TYPE ComplexStruct :
STRUCT
	intVal	:INT:=100;
	DintArr: ARRAY[1..5] OF DINT := [1, 2, 3, 4,100];
	BoolVal	:BOOL:= TRUE;
	ByteVal	:BYTE:=12;
	LrealVal	:LREAL:= 123.67;
	strVal 	:STRING(10):= 'hello';
	//strArray: ARRAY[1..3] OF STRING(10) := ['abc', 'qwe', 'hjk'];  ??
	SimpleStruct1		:SimpleStruct;	
END_STRUCT
END_TYPE

(* stored: Version 1.1.0.1, ProductVersion 3.1.4022.16
   DUT ComplexStruct: Id {15b4b77e-d9ed-4452-9369-ebc974ec09b9} *)
